{attribute 'GeneratedUsingTerminal: KL6211-0004'}
{attribute addProperty BoxType "KL6211-0004"}
{attribute addProperty Description ""}
{attribute addProperty Physics ""}
{attribute addProperty Id "Channel_1AT %Q*Channel_A6A8AB450"}
{attribute addProperty CRC "1899239057"}
{attribute addProperty Size "0"}
TYPE KL_71341691 :
STRUCT
	{attribute addProperty Name "Channel_1"}
	Channel_1 : Channel_A6A8AB45;
END_STRUCT
END_TYPE

(* stored: Version 1.2.0.0, ProductVersion 3.1.4024.9
   DUT KL_71341691: Id {3664bf33-f758-4b58-b32d-955bb953cb3a} *)
